// TIA Portal V20 export
DATA_BLOCK "instFB_ManualCtrl"   // DB
TITLE = instFB_ManualCtrl (Phase G)
VERSION : 1.1
// Phase G (C67, 2026-05-18) — instance DB for FB_ManualCtrl. Holds 4 MC_MoveJog + 1 MC_MoveLinearAbsolute + 1 R_TRIG + 1 Bool static. Total 6 multi-instance MC slots; with FB_AxisCtrl's 14 + FB_AutoCtrl_ABCDE's 1 = 21 declared system-wide, well under OB91 budget.
// stored: InstanceOfName FB_ManualCtrl, InstanceOfType FB
"FB_ManualCtrl"
   // VAR
   //    instJog_J1 { S7_SetPoint := 'True'} : MC_MOVEJOG;
   //    instJog_J2 { S7_SetPoint := 'True'} : MC_MOVEJOG;
   //    instJog_J3 { S7_SetPoint := 'True'} : MC_MOVEJOG;
   //    instJog_J4 { S7_SetPoint := 'True'} : MC_MOVEJOG;
   //    instMoveLinAbs : MC_MOVELINEARABSOLUTE;
   //    sRTRIGKinGo { S7_SetPoint := 'True'} : R_TRIG;
   //    statManualOK : Bool;
   //    statKinExecutePulse : Bool;
   // END_VAR
BEGIN
END_DATA_BLOCK
